INTERFACE I_Component
VAR_INPUT
END_VAR

VAR_OUTPUT
END_VAR

METHOD M_Disable : BOOL
VAR_INPUT
END_VAR
END_METHOD

METHOD M_Enable : BOOL
VAR_INPUT
END_VAR
END_METHOD

METHOD M_Halt : BOOL
VAR_INPUT
END_VAR
END_METHOD

METHOD M_Resume : BOOL
VAR_INPUT
END_VAR
END_METHOD

END_INTERFACE

(* stored: Version 1.1.0.1, ProductVersion 3.1.4024.15
   Itf I_Component: Id {3337d348-193e-4804-bc6d-8f5b2d280baf}
   Method M_Disable: Id {3f58ddfd-72fe-4d3d-b4d4-5870182f7e75}
   Method M_Enable: Id {209f0ab3-aef7-46f3-99d5-2c1e607ce3a0}
   Method M_Halt: Id {65f0acb6-737d-487e-a1b7-0fd6741c7d88}
   Method M_Resume: Id {f90a8a0b-dedc-4c7f-9fac-f4ef5a2a59aa} *)
